FUNCTION_BLOCK FB_EGBuero
VAR_INPUT
END_VAR
VAR_OUTPUT
END_VAR
VAR_IN_OUT
	
END_VAR
VAR
	bInit					: BOOL := TRUE;

  fbLichtBueroChef : FB_LichtBewegungsmelder;
  fbLichtBueroAssist : FB_LichtBewegungsmelder;
  fbLichtPausenraum : FB_LichtBewegungsmelder;

  bGruppeAus : bool;
	tKurz : TIME;
	tLang : TIME;
  
END_VAR


tKurz := DINT_TO_TIME(VnvdiLichtTofKurz * 60000);
tLang := DINT_TO_TIME(VnvdiLichtTofLang * 60000);
  
fbLichtBueroChef(
	tKurz:= tKurz, 
	tLang:= tLang, 
  bGruppeAus:= bGruppeAus,
	IOstTimeSwitchTimes:= VnvstSwitchTimesLichtBWMtofLang);
  
fbLichtBueroAssist(
	tKurz:= tKurz, 
	tLang:= tLang, 
  bGruppeAus:= bGruppeAus,
	IOstTimeSwitchTimes:= VnvstSwitchTimesLichtBWMtofLang);
  
fbLichtPausenraum(
	tKurz:= tKurz, 
	tLang:= tLang, 
  bGruppeAus:= bGruppeAus,
	IOstTimeSwitchTimes:= VnvstSwitchTimesLichtBWMtofLang);
  
  
(* FB END*)

END_FUNCTION_BLOCK

(* stored: Version 1.1.0.1, ProductVersion 3.1.4018.9
   POU FB_EGBuero: Id {1fd593b5-afbf-4a59-bd99-53e37dcca5fa}, SpecialFunc None *)
